VAR_GLOBAL
	Axis : ST_PosInterface;
END_VAR

(* stored: Version 1.1.0.1, ProductVersion 3.1.4024.3
   GVL GVL_IO: Id {2a792c51-4e91-457e-b510-83e13d39ffd9} *)
